# EPICS autosave request: iocBoot/gmca_23b_ioc2/dbSave/TV_V1_.req
%
% BURT Request File
%
% $(P)TV:V1:  High resolution camera
%

file assy.req ASSY=$(P)TV:V1
file mtr1.req MTR1=$(P)TV:mz1
file drv1.req DRV1=$(P)TV:ZM1
